Fanuc KAREL source: POST_ERR_L.kl

PROGRAM T
%NOLOCKGROUP
VAR
 v0 : INTEGER
 v1 : STRING[40]
 v2 : INTEGER
 v3 : INTEGER
BEGIN
 POST_ERR_L(v0, v1, v2, v3)
END T
